FUNCTION_BLOCK SL_Dose (* Dose contract: Requires NeedleDown AND VialPresent AND NOT Stoppered AND (P1 >= 0.1) AND (P1 <= 2.0); Ensures FilledMl >= TargetMl; Invariant NeedleDown AND VialPresent AND NOT Stoppered *)
  (* Standard: 61499-2 *)
  (* Version 2.0, 2026-09-27, Project contributors, Filling cell reference model *)
  PACKAGE fillingcell;
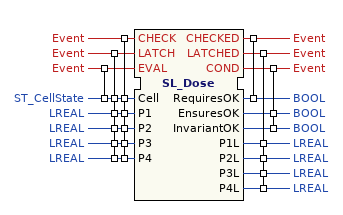
  EVENT_INPUT
    CHECK WITH Cell, P1, P2, P3, P4;
    LATCH WITH Cell, P1, P2, P3, P4;
    EVAL WITH Cell;
  END_EVENT
  EVENT_OUTPUT
    CHECKED WITH RequiresOK;
    LATCHED WITH P1L, P2L, P3L, P4L;
    COND WITH EnsuresOK, InvariantOK;
  END_EVENT
  VAR_INPUT
    Cell : fillingcell::ST_CellState;
    P1 : LREAL;
    P2 : LREAL;
    P3 : LREAL;
    P4 : LREAL;
  END_VAR
  VAR_OUTPUT
    RequiresOK : BOOL;
    EnsuresOK : BOOL;
    InvariantOK : BOOL;
    P1L : LREAL;
    P2L : LREAL;
    P3L : LREAL;
    P4L : LREAL;
  END_VAR
  VAR
    TargetMl : LREAL;
  END_VAR
  EC_STATES
    CHECK : CHECK -> CHECKED;
    LATCH : LATCH -> LATCHED;
    EVAL : EVAL -> COND;
  END_STATES
  ALGORITHM CHECK IN ST:
RequiresOK := Cell.Valid AND Cell.Safe AND (Cell.NeedleDown AND Cell.VialPresent AND NOT Cell.Stoppered AND (P1 >= 0.1) AND (P1 <= 2.0));
  END_ALGORITHM
  ALGORITHM LATCH IN ST:
P1L := P1;
P2L := P2;
P3L := P3;
P4L := P4;
TargetMl := Cell.FilledMl + P1;
  END_ALGORITHM
  ALGORITHM EVAL IN ST:
EnsuresOK := Cell.FilledMl >= TargetMl;
InvariantOK := Cell.Valid AND Cell.Safe AND (Cell.NeedleDown AND Cell.VialPresent AND NOT Cell.Stoppered);
  END_ALGORITHM
END_FUNCTION_BLOCK
